TYPE ST_CameraData :
STRUCT
	CurrentJobID			: WORD;
	ErrorCode				: WORD;
	AcquisitionID			: WORD;
	InspectionID			: WORD;
	InspectionResultCode	: WORD;
	Results					: ST_CameraResults;
END_STRUCT
END_TYPE

(* stored: Version 1.1.0.1, ProductVersion 3.1.4024.9
   DUT ST_CameraData: Id {941eca32-b1aa-4f17-89b6-6939c90deac4} *)
